Staubli VAL3: listFilling.pgx

public program listFilling(num x_nListNumber, string& x_sItemList[], num& x_nError)
  local num l_nI
begin

  // This program fills a list object with items

  //

  // Input Param

  //  x_nListNumber  : list number to fill

  //  x_sItemList    : Items to push into the List object

  //

  // Output Param

  //  x_Error : Error code

  //          = 3    : Variable sListItemX doesn't exist

  //

  //--------------------------------------------------------------

  //

  x_nError=0

  switch x_nListNumber

    case 0

      resize(sListItem0,1,size(x_sItemList))

      for l_nI=0 to size(x_sItemList)-1

        sListItem0[l_nI]=x_sItemList[l_nI]

      endFor

    break

    default

      x_nError=3

    break

  endSwitch

  //

end
